// TIA Portal V19 export
FUNCTION "LOmacAPcFr_StartupConfiguration" : Void   // FC39, LAD
{ S7_Optimized_Access := 'TRUE' }
// stored: SetENOAutomatically false
   VAR_OUTPUT
      configurationOmac : "typeLPMLV30_Configuration";
      configurationLanguage : Int;
   END_VAR
   VAR_TEMP
      tempIndex : Int;
      tempLocalSC : Bool;   // State complete signal (one cycle)
   END_VAR
   VAR_TEMP   // added for the SCL form of the ladder/FBD networks
      _w1 : Bool;
      _w2 : Bool;
   END_VAR
BEGIN

REGION Network 1: Mode configuration
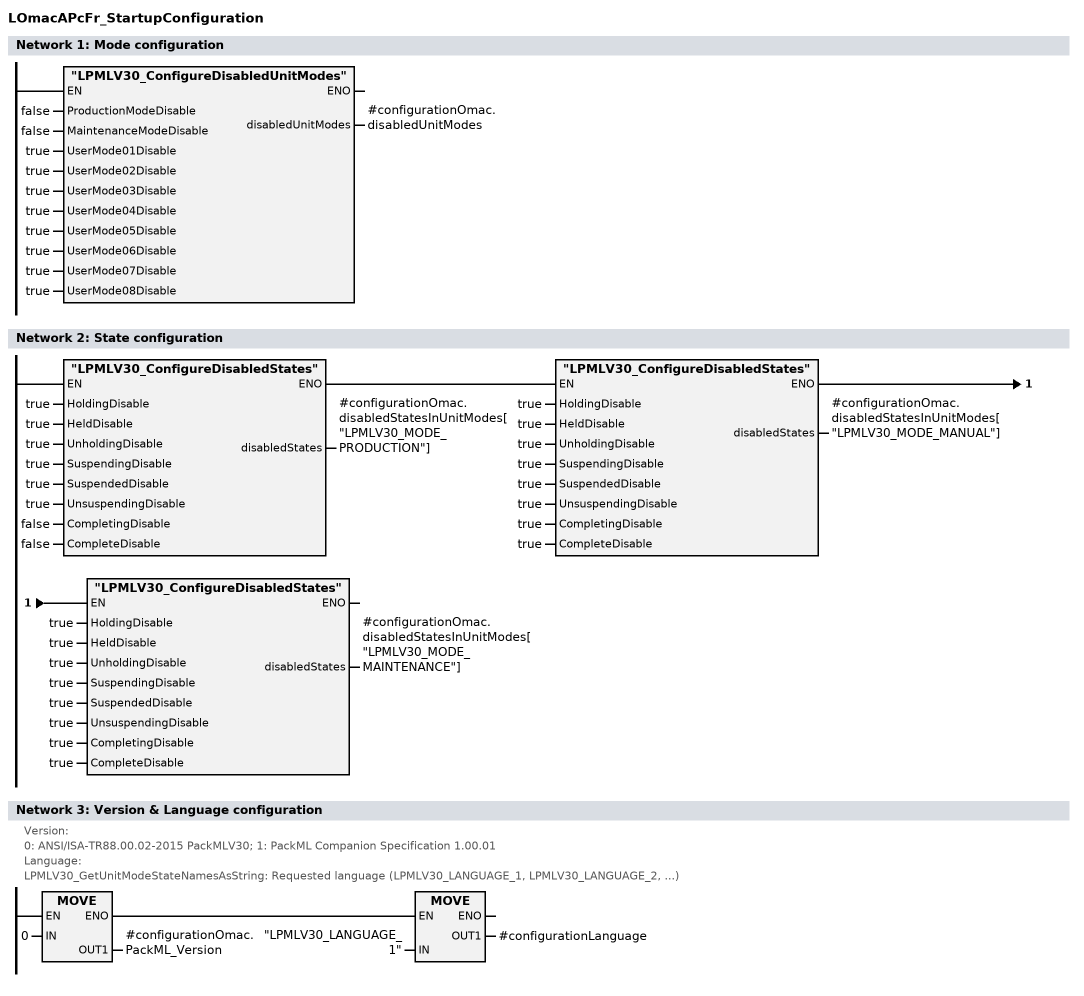
   RUNG wire#powerrail
      "LPMLV30_ConfigureDisabledUnitModes"(ProductionModeDisable := false, MaintenanceModeDisable := false, UserMode01Disable := true, UserMode02Disable := true, UserMode03Disable := true, UserMode04Disable := true, UserMode05Disable := true, UserMode06Disable := true, UserMode07Disable := true, UserMode08Disable := true, disabledUnitModes => #configurationOmac.disabledUnitModes)
   END_RUNG
   // the same network as SCL:
   "LPMLV30_ConfigureDisabledUnitModes"(ProductionModeDisable := false,
                           MaintenanceModeDisable := false,
                           UserMode01Disable := true,
                           UserMode02Disable := true,
                           UserMode03Disable := true,
                           UserMode04Disable := true,
                           UserMode05Disable := true,
                           UserMode06Disable := true,
                           UserMode07Disable := true,
                           UserMode08Disable := true,
                           disabledUnitModes => #configurationOmac.disabledUnitModes);
END_REGION

REGION Network 2: State configuration
   RUNG wire#powerrail
      "LPMLV30_ConfigureDisabledStates"(HoldingDisable := true, HeldDisable := true, UnholdingDisable := true, SuspendingDisable := true, SuspendedDisable := true, UnsuspendingDisable := true, CompletingDisable := false, CompleteDisable := false, disabledStates => #configurationOmac.disabledStatesInUnitModes["LPMLV30_MODE_PRODUCTION"])
      "LPMLV30_ConfigureDisabledStates"(HoldingDisable := true, HeldDisable := true, UnholdingDisable := true, SuspendingDisable := true, SuspendedDisable := true, UnsuspendingDisable := true, CompletingDisable := true, CompleteDisable := true, disabledStates => #configurationOmac.disabledStatesInUnitModes["LPMLV30_MODE_MANUAL"])
      "LPMLV30_ConfigureDisabledStates"(HoldingDisable := true, HeldDisable := true, UnholdingDisable := true, SuspendingDisable := true, SuspendedDisable := true, UnsuspendingDisable := true, CompletingDisable := true, CompleteDisable := true, disabledStates => #configurationOmac.disabledStatesInUnitModes["LPMLV30_MODE_MAINTENANCE"])
   END_RUNG
   // the same network as SCL:
   "LPMLV30_ConfigureDisabledStates"(HoldingDisable := true,
                           HeldDisable := true,
                           UnholdingDisable := true,
                           SuspendingDisable := true,
                           SuspendedDisable := true,
                           UnsuspendingDisable := true,
                           CompletingDisable := false,
                           CompleteDisable := false,
                           disabledStates => #configurationOmac.disabledStatesInUnitModes["LPMLV30_MODE_PRODUCTION"],
                           ENO => #_w1);
   "LPMLV30_ConfigureDisabledStates"(EN := #_w1,
                           HoldingDisable := true,
                           HeldDisable := true,
                           UnholdingDisable := true,
                           SuspendingDisable := true,
                           SuspendedDisable := true,
                           UnsuspendingDisable := true,
                           CompletingDisable := true,
                           CompleteDisable := true,
                           disabledStates => #configurationOmac.disabledStatesInUnitModes["LPMLV30_MODE_MANUAL"],
                           ENO => #_w2);
   IF #_w2 THEN
       "LPMLV30_ConfigureDisabledStates"(HoldingDisable := true,
                               HeldDisable := true,
                               UnholdingDisable := true,
                               SuspendingDisable := true,
                               SuspendedDisable := true,
                               UnsuspendingDisable := true,
                               CompletingDisable := true,
                               CompleteDisable := true,
                               disabledStates => #configurationOmac.disabledStatesInUnitModes["LPMLV30_MODE_MAINTENANCE"]);
   END_IF;
END_REGION

REGION Network 3: Version & Language configuration
   // Version:
   // 0: ANSI/ISA-TR88.00.02-2015 PackMLV30; 1: PackML Companion Specification 1.00.01
   // 
   // Language:
   // LPMLV30_GetUnitModeStateNamesAsString: Requested language (LPMLV30_LANGUAGE_1, LPMLV30_LANGUAGE_2, ...)
   RUNG wire#powerrail
      Move(in := 0, out1 => #configurationOmac.PackML_Version)
      Move(in := "LPMLV30_LANGUAGE_1", out1 => #configurationLanguage)
   END_RUNG
   // the same network as SCL:
   #configurationOmac.PackML_Version := 0;
   #configurationLanguage := "LPMLV30_LANGUAGE_1";
END_REGION
END_FUNCTION
